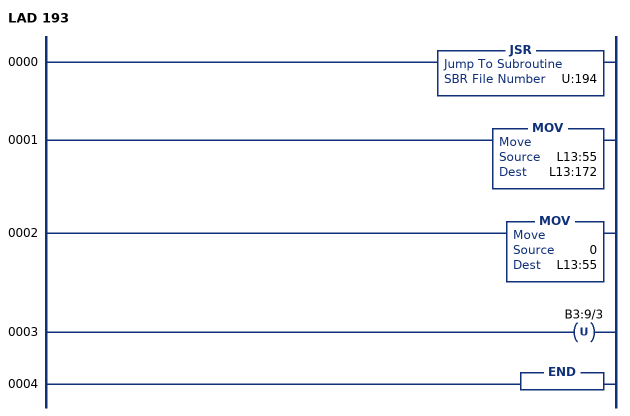
% Rung: 0 %
SOR JSR U:194 EOR
% Rung: 1 %
SOR MOV L13:55 L13:172 EOR
% Rung: 2 %
SOR MOV 0 L13:55 EOR
% Rung: 3 %
SOR OTU B3:9/3 EOR
% Rung: 4 %
SOR END EOR

LADDER 194
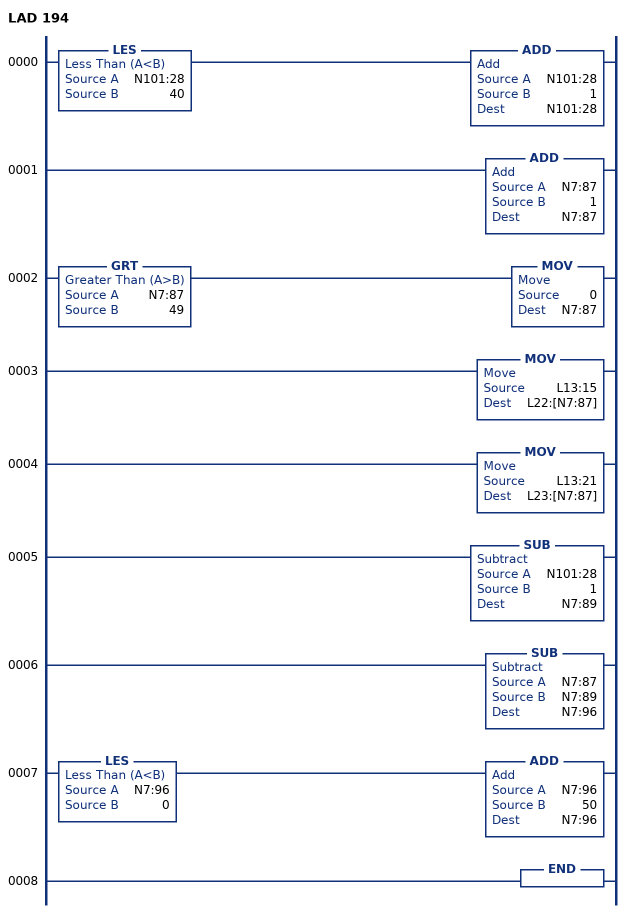
% Rung: 0 %
SOR LES N101:28 40 ADD N101:28 1 N101:28 EOR
% Rung: 1 %
SOR ADD N7:87 1 N7:87 EOR
% Rung: 2 %
SOR GRT N7:87 49 MOV 0 N7:87 EOR
% Rung: 3 %
SOR MOV L13:15 L22:[N7:87] EOR
% Rung: 4 %
SOR MOV L13:21 L23:[N7:87] EOR
% Rung: 5 %
SOR SUB N101:28 1 N7:89 EOR
% Rung: 6 %
SOR SUB N7:87 N7:89 N7:96 EOR
% Rung: 7 %
SOR LES N7:96 0 ADD N7:96 50 N7:96 EOR
% Rung: 8 %
SOR END EOR

LADDER 195
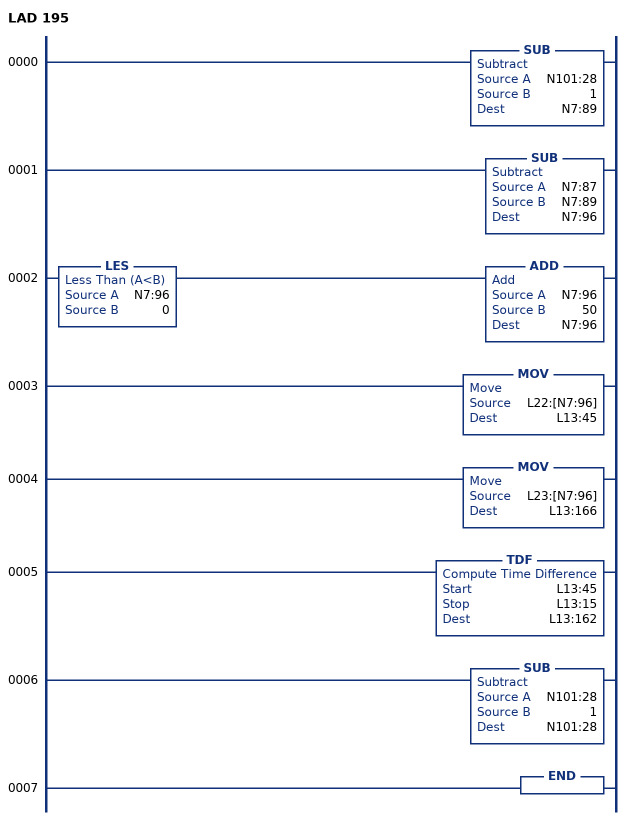
% Rung: 0 %
SOR SUB N101:28 1 N7:89 EOR
% Rung: 1 %
SOR SUB N7:87 N7:89 N7:96 EOR
% Rung: 2 %
SOR LES N7:96 0 ADD N7:96 50 N7:96 EOR
% Rung: 3 %
SOR MOV L22:[N7:96] L13:45 EOR
% Rung: 4 %
SOR MOV L23:[N7:96] L13:166 EOR
% Rung: 5 %
SOR TDF L13:45 L13:15 L13:162 EOR
% Rung: 6 %
SOR SUB N101:28 1 N101:28 EOR
% Rung: 7 %
SOR END EOR

LADDER 196
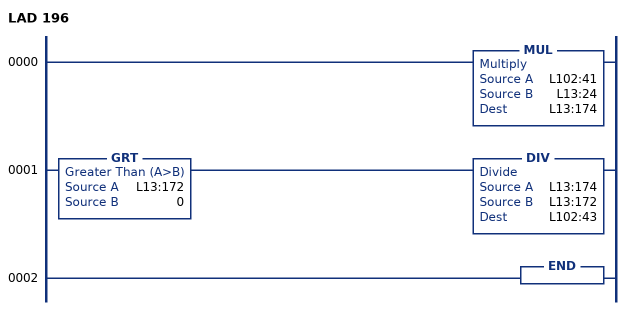
% Rung: 0 %
SOR MUL L102:41 L13:24 L13:174 EOR
% Rung: 1 %
SOR GRT L13:172 0 DIV L13:174 L13:172 L102:43 EOR
% Rung: 2 %
SOR END EOR

LADDER 197
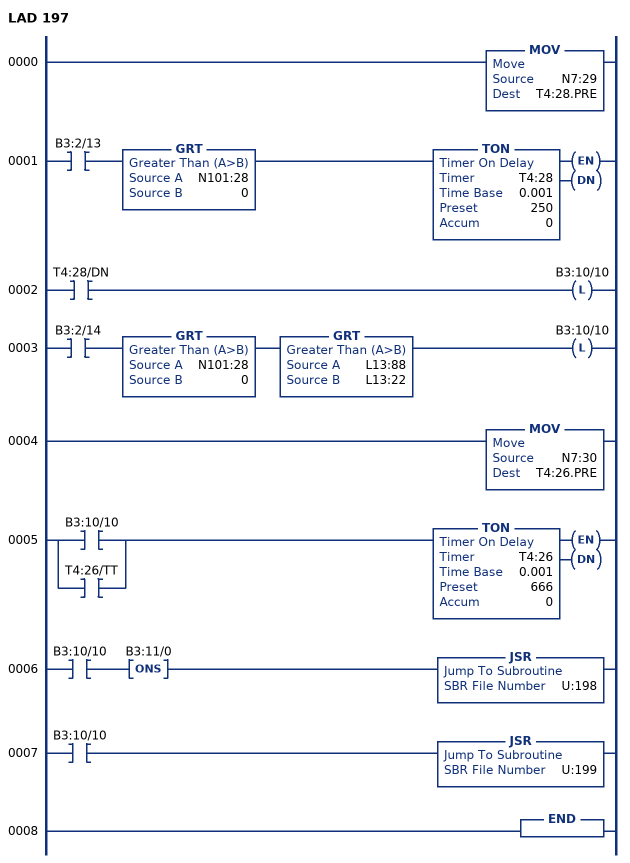
% Rung: 0 %
SOR MOV N7:29 T4:28.PRE EOR
% Rung: 1 %
SOR XIC B3:2/13 GRT N101:28 0 TON T4:28 0.001 250 0 EOR
% Rung: 2 %
SOR XIC T4:28/DN OTL B3:10/10 EOR
% Rung: 3 %
SOR XIC B3:2/14 GRT N101:28 0 GRT L13:88 L13:22 OTL B3:10/10 EOR
% Rung: 4 %
SOR MOV N7:30 T4:26.PRE EOR
% Rung: 5 %
SOR BST XIC B3:10/10 NXB XIC T4:26/TT BND TON T4:26 0.001 666 0 EOR
% Rung: 6 %
SOR XIC B3:10/10 ONS B3:11/0 JSR U:198 EOR
% Rung: 7 %
SOR XIC B3:10/10 JSR U:199 EOR
% Rung: 8 %
SOR END EOR

LADDER 198
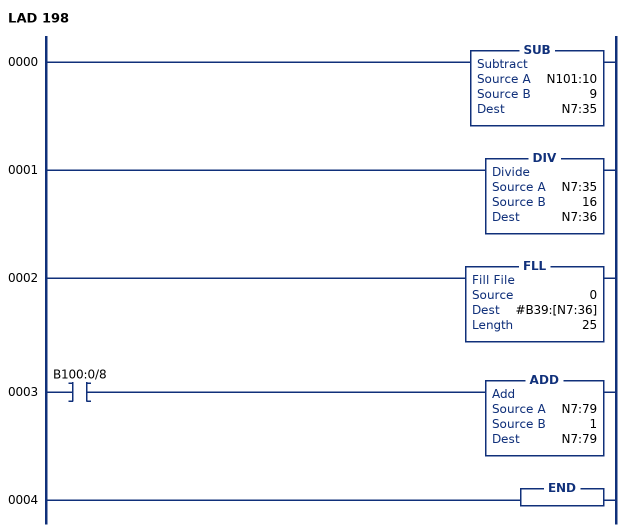
% Rung: 0 %
SOR SUB N101:10 9 N7:35 EOR
% Rung: 1 %
SOR DIV N7:35 16 N7:36 EOR
% Rung: 2 %
SOR FLL 0 #B39:[N7:36] 25 EOR
% Rung: 3 %
SOR XIC B100:0/8 ADD N7:79 1 N7:79 EOR
% Rung: 4 %
SOR END EOR

LADDER 199
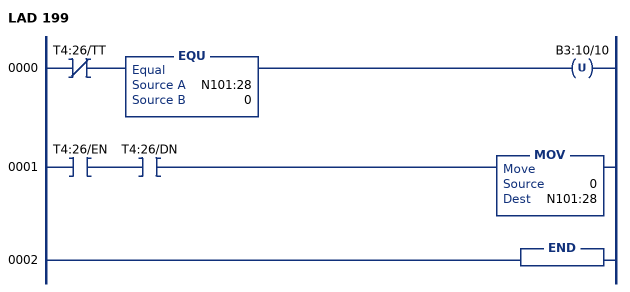
% Rung: 0 %
SOR XIO T4:26/TT EQU N101:28 0 OTU B3:10/10 EOR
% Rung: 1 %
SOR XIC T4:26/EN XIC T4:26/DN MOV 0 N101:28 EOR
% Rung: 2 %
SOR END EOR

LADDER 200
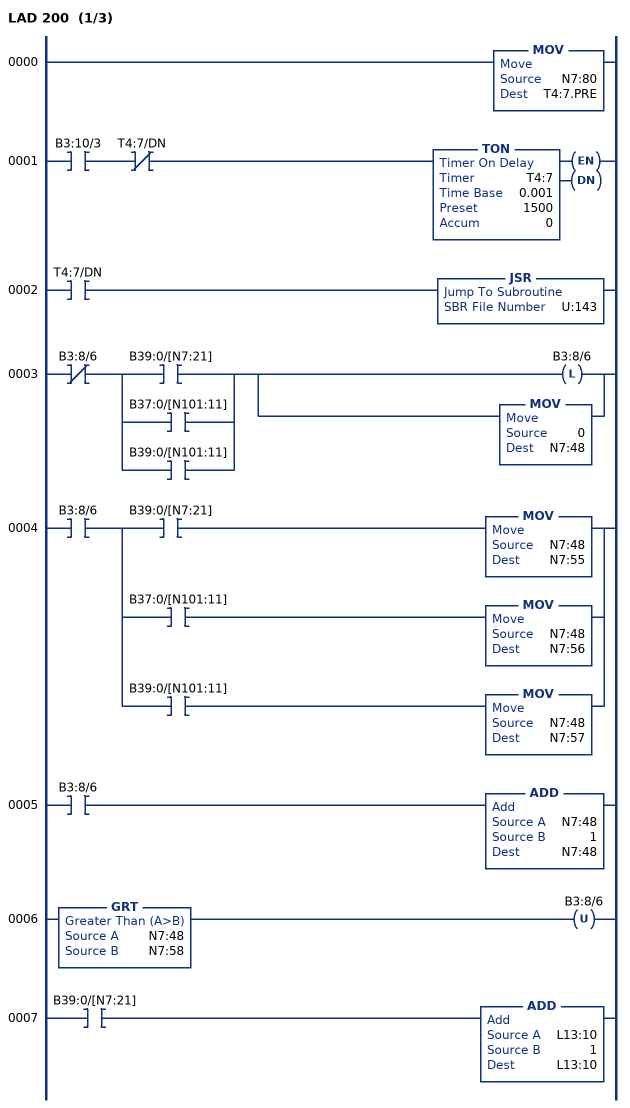
% Rung: 0 %
SOR MOV N7:80 T4:7.PRE EOR
% Rung: 1 %
SOR XIC B3:10/3 XIO T4:7/DN TON T4:7 0.001 1500 0 EOR
% Rung: 2 %
SOR XIC T4:7/DN JSR U:143 EOR
% Rung: 3 %
SOR XIO B3:8/6 BST XIC B39:0/[N7:21] NXB XIC B37:0/[N101:11] NXB XIC B39:0/[N101:11] BND BST OTL B3:8/6 NXB MOV 0 N7:48 BND EOR
% Rung: 4 %
SOR XIC B3:8/6 BST XIC B39:0/[N7:21] MOV N7:48 N7:55 NXB XIC B37:0/[N101:11] MOV N7:48 N7:56 NXB XIC B39:0/[N101:11] MOV N7:48 N7:57 BND EOR
% Rung: 5 %
SOR XIC B3:8/6 ADD N7:48 1 N7:48 EOR
% Rung: 6 %
SOR GRT N7:48 N7:58 OTU B3:8/6 EOR
% Rung: 7 %
SOR XIC B39:0/[N7:21] ADD L13:10 1 L13:10 EOR

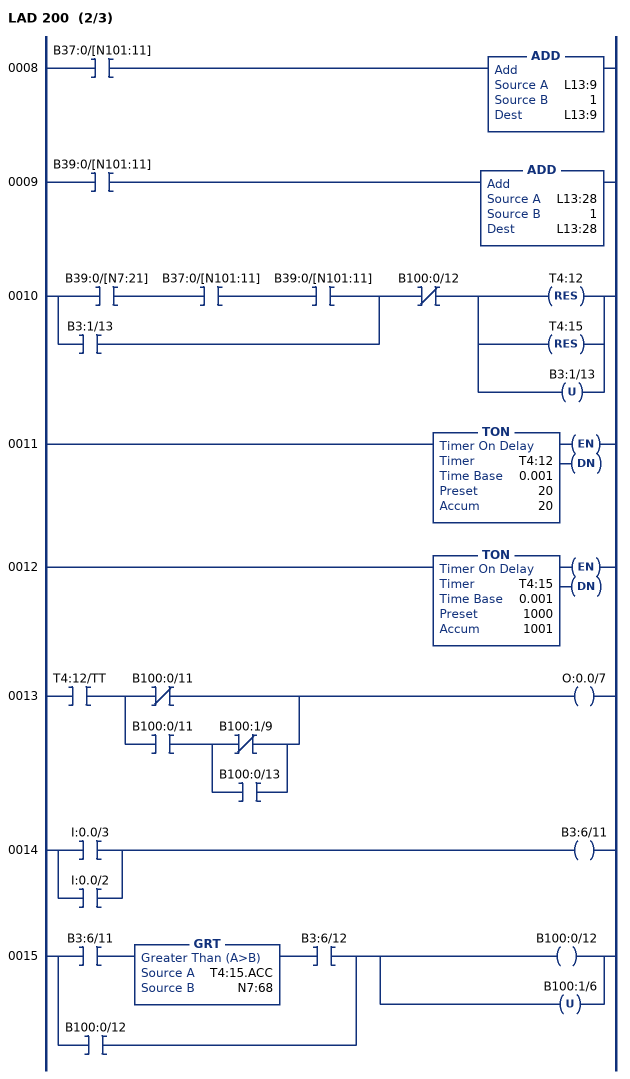
% Rung: 8 %
SOR XIC B37:0/[N101:11] ADD L13:9 1 L13:9 EOR
% Rung: 9 %
SOR XIC B39:0/[N101:11] ADD L13:28 1 L13:28 EOR
% Rung: 10 %
SOR BST XIC B39:0/[N7:21] XIC B37:0/[N101:11] XIC B39:0/[N101:11] NXB XIC B3:1/13 BND XIO B100:0/12 BST RES T4:12 NXB RES T4:15 NXB OTU B3:1/13 BND EOR
% Rung: 11 %
SOR TON T4:12 0.001 20 20 EOR
% Rung: 12 %
SOR TON T4:15 0.001 1000 1001 EOR
% Rung: 13 %
SOR XIC T4:12/TT BST XIO B100:0/11 NXB XIC B100:0/11 BST XIO B100:1/9 NXB XIC B100:0/13 BND BND OTE O:0.0/7 EOR
% Rung: 14 %
SOR BST XIC I:0.0/3 NXB XIC I:0.0/2 BND OTE B3:6/11 EOR
% Rung: 15 %
SOR BST XIC B3:6/11 GRT T4:15.ACC N7:68 XIC B3:6/12 NXB XIC B100:0/12 BND BST OTE B100:0/12 NXB OTU B100:1/6 BND EOR

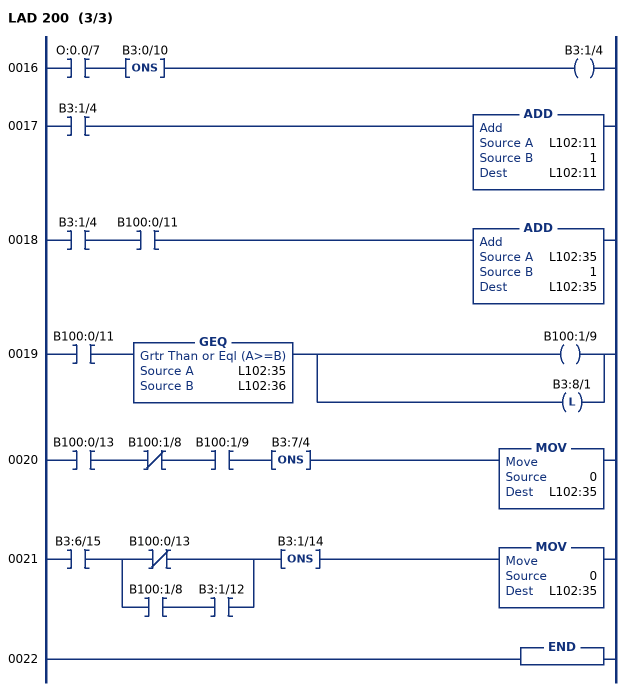
% Rung: 16 %
SOR XIC O:0.0/7 ONS B3:0/10 OTE B3:1/4 EOR
% Rung: 17 %
SOR XIC B3:1/4 ADD L102:11 1 L102:11 EOR
% Rung: 18 %
SOR XIC B3:1/4 XIC B100:0/11 ADD L102:35 1 L102:35 EOR
% Rung: 19 %
SOR XIC B100:0/11 GEQ L102:35 L102:36 BST OTE B100:1/9 NXB OTL B3:8/1 BND EOR
% Rung: 20 %
SOR XIC B100:0/13 XIO B100:1/8 XIC B100:1/9 ONS B3:7/4 MOV 0 L102:35 EOR
% Rung: 21 %
SOR XIC B3:6/15 BST XIO B100:0/13 NXB XIC B100:1/8 XIC B3:1/12 BND ONS B3:1/14 MOV 0 L102:35 EOR
% Rung: 22 %
SOR END EOR

LADDER 235
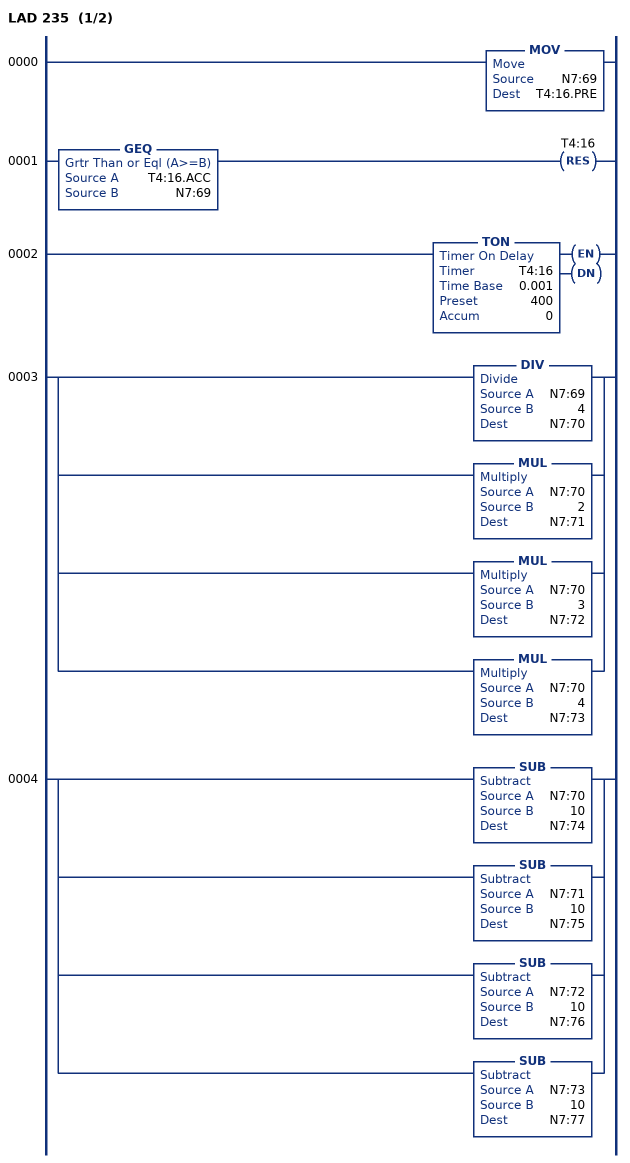
% Rung: 0 %
SOR MOV N7:69 T4:16.PRE EOR
% Rung: 1 %
SOR GEQ T4:16.ACC N7:69 RES T4:16 EOR
% Rung: 2 %
SOR TON T4:16 0.001 400 0 EOR
% Rung: 3 %
SOR BST DIV N7:69 4 N7:70 NXB MUL N7:70 2 N7:71 NXB MUL N7:70 3 N7:72 NXB MUL N7:70 4 N7:73 BND EOR
% Rung: 4 %
SOR BST SUB N7:70 10 N7:74 NXB SUB N7:71 10 N7:75 NXB SUB N7:72 10 N7:76 NXB SUB N7:73 10 N7:77 BND EOR

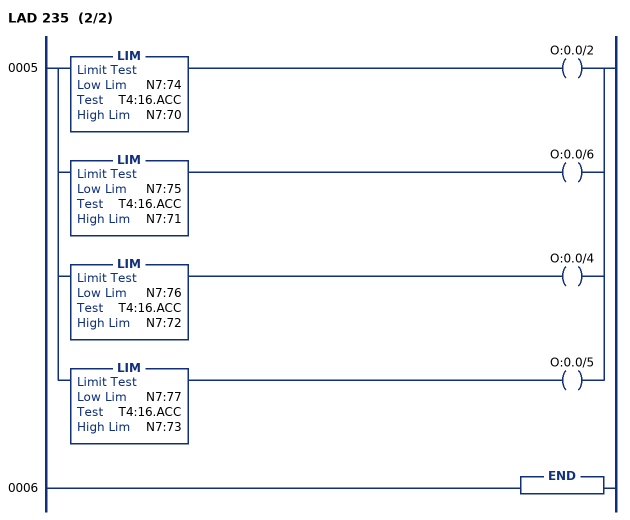
% Rung: 5 %
SOR BST LIM N7:74 T4:16.ACC N7:70 OTE O:0.0/2 NXB LIM N7:75 T4:16.ACC N7:71 OTE O:0.0/6 NXB LIM N7:76 T4:16.ACC N7:72 OTE O:0.0/4 NXB LIM N7:77 T4:16.ACC N7:73 OTE O:0.0/5 BND EOR
% Rung: 6 %
SOR END EOR

LADDER 236
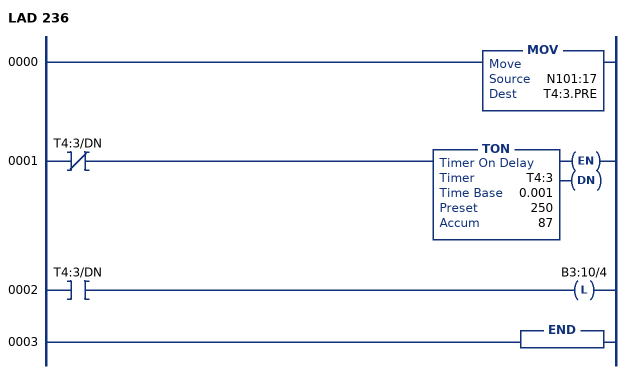
% Rung: 0 %
SOR MOV N101:17 T4:3.PRE EOR
% Rung: 1 %
SOR XIO T4:3/DN TON T4:3 0.001 250 87 EOR
% Rung: 2 %
SOR XIC T4:3/DN OTL B3:10/4 EOR
% Rung: 3 %
SOR END EOR

LADDER 237
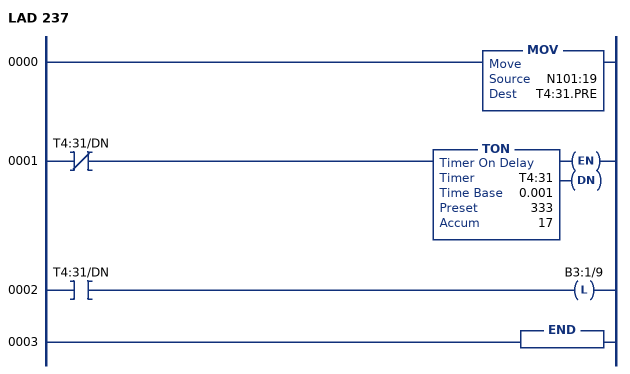
% Rung: 0 %
SOR MOV N101:19 T4:31.PRE EOR
% Rung: 1 %
SOR XIO T4:31/DN TON T4:31 0.001 333 17 EOR
% Rung: 2 %
SOR XIC T4:31/DN OTL B3:1/9 EOR
% Rung: 3 %
SOR END EOR

LADDER 238
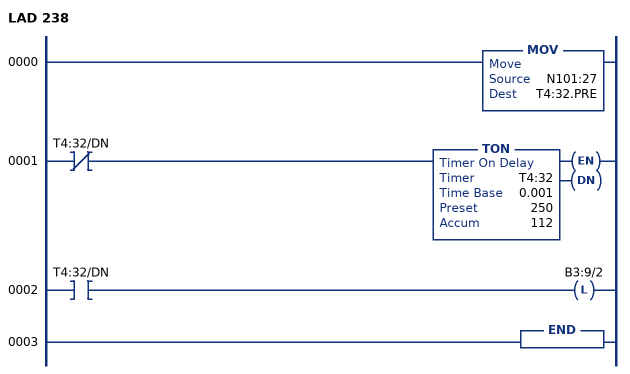
% Rung: 0 %
SOR MOV N101:27 T4:32.PRE EOR
% Rung: 1 %
SOR XIO T4:32/DN TON T4:32 0.001 250 112 EOR
% Rung: 2 %
SOR XIC T4:32/DN OTL B3:9/2 EOR
% Rung: 3 %
SOR END EOR

LADDER 239
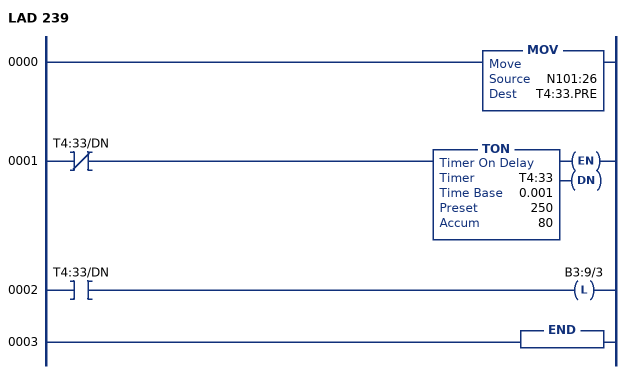
% Rung: 0 %
SOR MOV N101:26 T4:33.PRE EOR
% Rung: 1 %
SOR XIO T4:33/DN TON T4:33 0.001 250 80 EOR
% Rung: 2 %
SOR XIC T4:33/DN OTL B3:9/3 EOR
% Rung: 3 %
SOR END EOR

LADDER 240
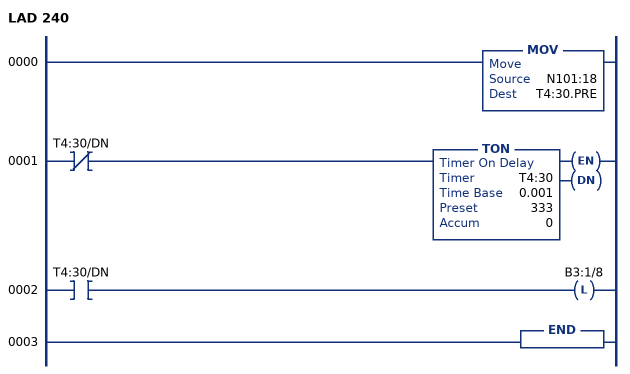
% Rung: 0 %
SOR MOV N101:18 T4:30.PRE EOR
% Rung: 1 %
SOR XIO T4:30/DN TON T4:30 0.001 333 0 EOR
% Rung: 2 %
SOR XIC T4:30/DN OTL B3:1/8 EOR
% Rung: 3 %
SOR END EOR

LADDER 241
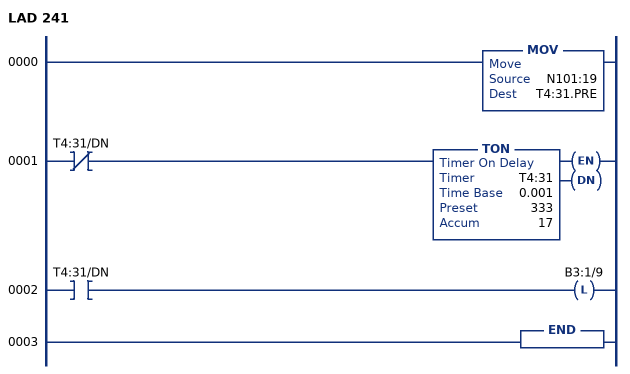
% Rung: 0 %
SOR MOV N101:19 T4:31.PRE EOR
% Rung: 1 %
SOR XIO T4:31/DN TON T4:31 0.001 333 17 EOR
% Rung: 2 %
SOR XIC T4:31/DN OTL B3:1/9 EOR
% Rung: 3 %
SOR END EOR

LADDER 242
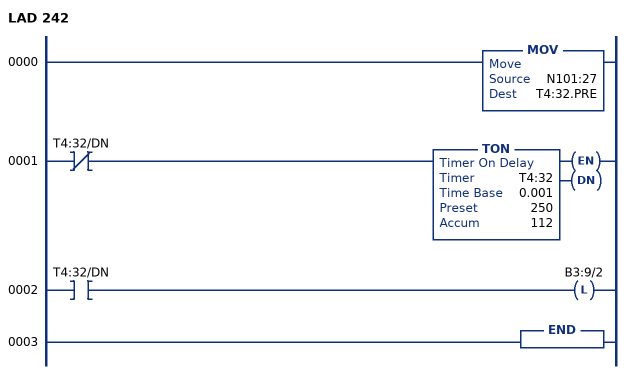
% Rung: 0 %
SOR MOV N101:27 T4:32.PRE EOR
% Rung: 1 %
SOR XIO T4:32/DN TON T4:32 0.001 250 112 EOR
% Rung: 2 %
SOR XIC T4:32/DN OTL B3:9/2 EOR
% Rung: 3 %
SOR END EOR

LADDER 243
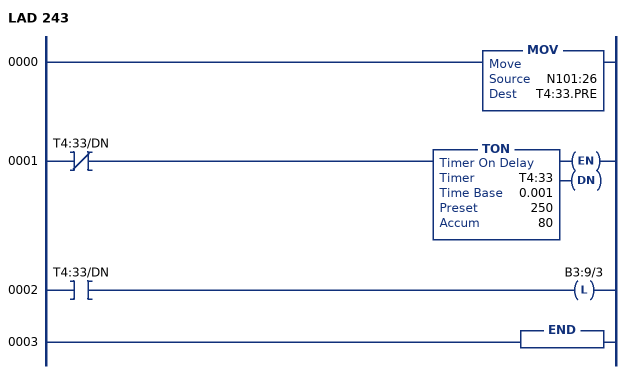
% Rung: 0 %
SOR MOV N101:26 T4:33.PRE EOR
% Rung: 1 %
SOR XIO T4:33/DN TON T4:33 0.001 250 80 EOR
% Rung: 2 %
SOR XIC T4:33/DN OTL B3:9/3 EOR
% Rung: 3 %
SOR END EOR

LADDER 244
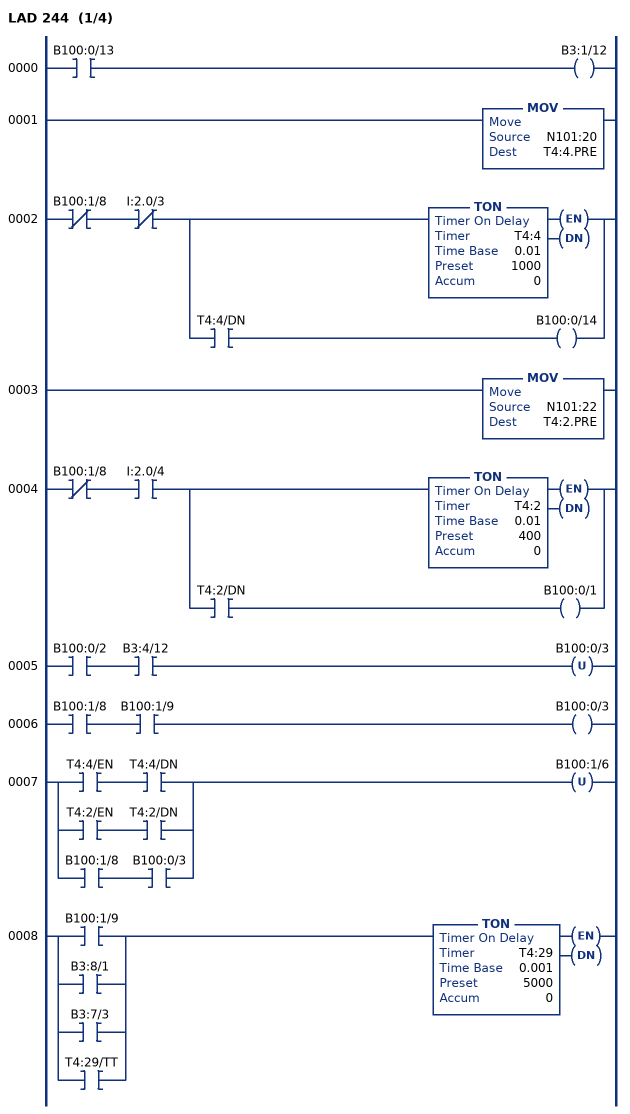
% Rung: 0 %
SOR XIC B100:0/13 OTE B3:1/12 EOR
% Rung: 1 %
SOR MOV N101:20 T4:4.PRE EOR
% Rung: 2 %
SOR XIO B100:1/8 XIO I:2.0/3 BST TON T4:4 0.01 1000 0 NXB XIC T4:4/DN OTE B100:0/14 BND EOR
% Rung: 3 %
SOR MOV N101:22 T4:2.PRE EOR
% Rung: 4 %
SOR XIO B100:1/8 XIC I:2.0/4 BST TON T4:2 0.01 400 0 NXB XIC T4:2/DN OTE B100:0/1 BND EOR
% Rung: 5 %
SOR XIC B100:0/2 XIC B3:4/12 OTU B100:0/3 EOR
% Rung: 6 %
SOR XIC B100:1/8 XIC B100:1/9 OTE B100:0/3 EOR
% Rung: 7 %
SOR BST XIC T4:4/EN XIC T4:4/DN NXB XIC T4:2/EN XIC T4:2/DN NXB XIC B100:1/8 XIC B100:0/3 BND OTU B100:1/6 EOR
% Rung: 8 %
SOR BST XIC B100:1/9 NXB XIC B3:8/1 NXB XIC B3:7/3 NXB XIC T4:29/TT BND TON T4:29 0.001 5000 0 EOR

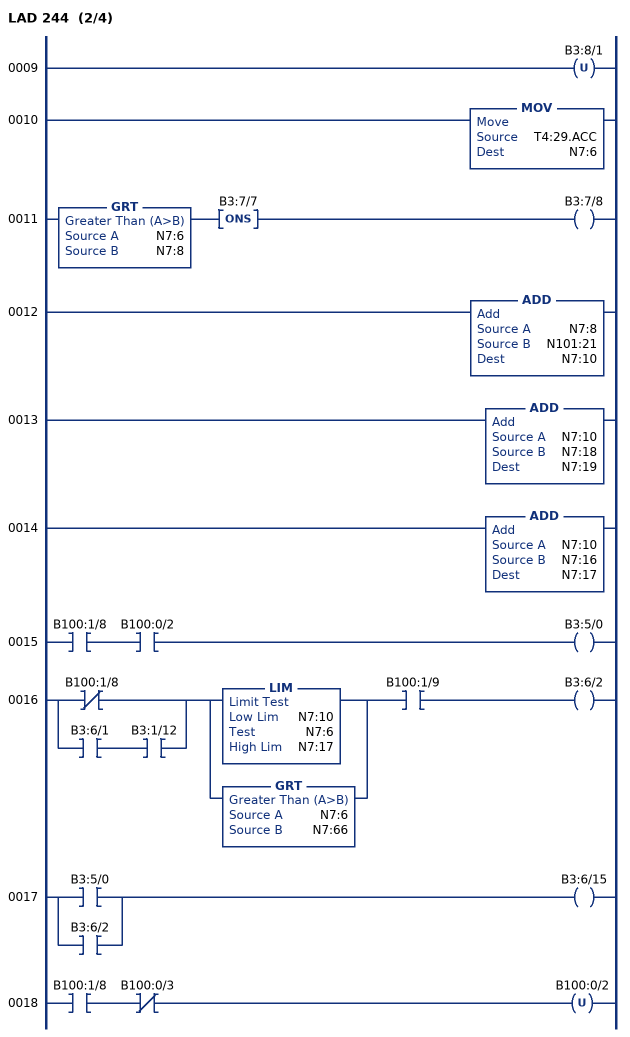
% Rung: 9 %
SOR OTU B3:8/1 EOR
% Rung: 10 %
SOR MOV T4:29.ACC N7:6 EOR
% Rung: 11 %
SOR GRT N7:6 N7:8 ONS B3:7/7 OTE B3:7/8 EOR
% Rung: 12 %
SOR ADD N7:8 N101:21 N7:10 EOR
% Rung: 13 %
SOR ADD N7:10 N7:18 N7:19 EOR
% Rung: 14 %
SOR ADD N7:10 N7:16 N7:17 EOR
% Rung: 15 %
SOR XIC B100:1/8 XIC B100:0/2 OTE B3:5/0 EOR
% Rung: 16 %
SOR BST XIO B100:1/8 NXB XIC B3:6/1 XIC B3:1/12 BND BST LIM N7:10 N7:6 N7:17 NXB GRT N7:6 N7:66 BND XIC B100:1/9 OTE B3:6/2 EOR
% Rung: 17 %
SOR BST XIC B3:5/0 NXB XIC B3:6/2 BND OTE B3:6/15 EOR
% Rung: 18 %
SOR XIC B100:1/8 XIO B100:0/3 OTU B100:0/2 EOR

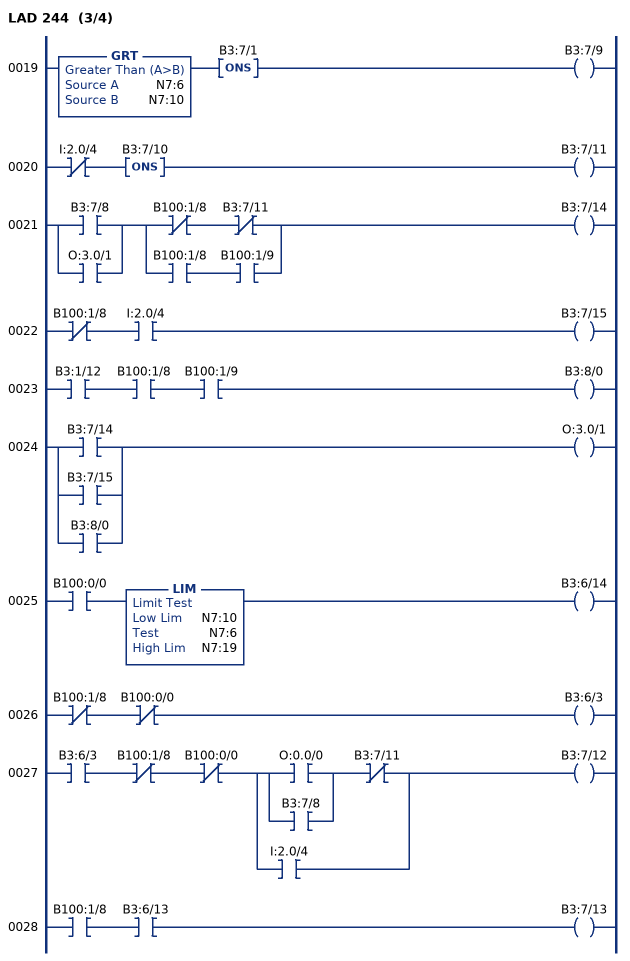
% Rung: 19 %
SOR GRT N7:6 N7:10 ONS B3:7/1 OTE B3:7/9 EOR
% Rung: 20 %
SOR XIO I:2.0/4 ONS B3:7/10 OTE B3:7/11 EOR
% Rung: 21 %
SOR BST XIC B3:7/8 NXB XIC O:3.0/1 BND BST XIO B100:1/8 XIO B3:7/11 NXB XIC B100:1/8 XIC B100:1/9 BND OTE B3:7/14 EOR
% Rung: 22 %
SOR XIO B100:1/8 XIC I:2.0/4 OTE B3:7/15 EOR
% Rung: 23 %
SOR XIC B3:1/12 XIC B100:1/8 XIC B100:1/9 OTE B3:8/0 EOR
% Rung: 24 %
SOR BST XIC B3:7/14 NXB XIC B3:7/15 NXB XIC B3:8/0 BND OTE O:3.0/1 EOR
% Rung: 25 %
SOR XIC B100:0/0 LIM N7:10 N7:6 N7:19 OTE B3:6/14 EOR
% Rung: 26 %
SOR XIO B100:1/8 XIO B100:0/0 OTE B3:6/3 EOR
% Rung: 27 %
SOR XIC B3:6/3 XIO B100:1/8 XIO B100:0/0 BST BST XIC O:0.0/0 NXB XIC B3:7/8 BND XIO B3:7/11 NXB XIC I:2.0/4 BND OTE B3:7/12 EOR
% Rung: 28 %
SOR XIC B100:1/8 XIC B3:6/13 OTE B3:7/13 EOR

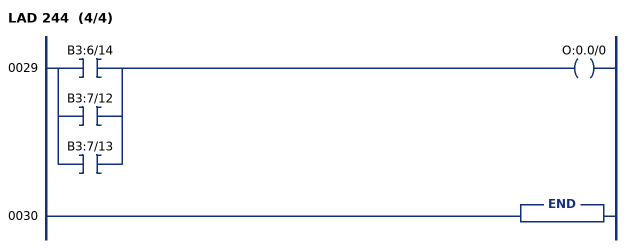
% Rung: 29 %
SOR BST XIC B3:6/14 NXB XIC B3:7/12 NXB XIC B3:7/13 BND OTE O:0.0/0 EOR
% Rung: 30 %
SOR END EOR

LADDER 245
